FUNCTION_BLOCK IA_GBSD (* ISOBUS Adapter for Ground Based Speed and Distance (GBSD) *)
  (* Standard: ISO 11783-7; Classification: PGN 65097; Description: Copyright (c) 2024-2026 HR Agrartechnik GmbH This program and the accompanying materials are made available under the terms of the Eclipse Public License 2.0 which is available at https://www.eclipse.org/legal/epl-2.0/ SPDX-License-Identifier: EPL-2.0 *)
  (* Version 1.0, 2026-04-19, Franz Höpfinger, HR Agrartechnik GmbH, initial API and implementation (Adapter Wrapper for I_GBSD) *)
  PACKAGE isobus::tecu;
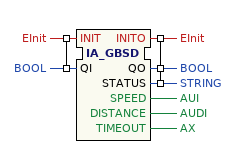
  EVENT_INPUT
    INIT : EInit WITH QI; (* Service Initialization *)
  END_EVENT
  EVENT_OUTPUT
    INITO : EInit WITH QO, STATUS; (* Initialization Confirm *)
  END_EVENT
  VAR_INPUT
    QI : BOOL; (* Event Input Qualifier *)
  END_VAR
  VAR_OUTPUT
    QO : BOOL; (* Event Output Qualifier *)
    STATUS : STRING;
  END_VAR
  PLUGS
    SPEED : adapter::types::unidirectional::AUI; (* Ground-based machine speed *)
    DISTANCE : adapter::types::unidirectional::AUDI; (* Ground-based machine distance *)
    TIMEOUT : adapter::types::unidirectional::AX; (* Timeout Status *)
  END_PLUGS
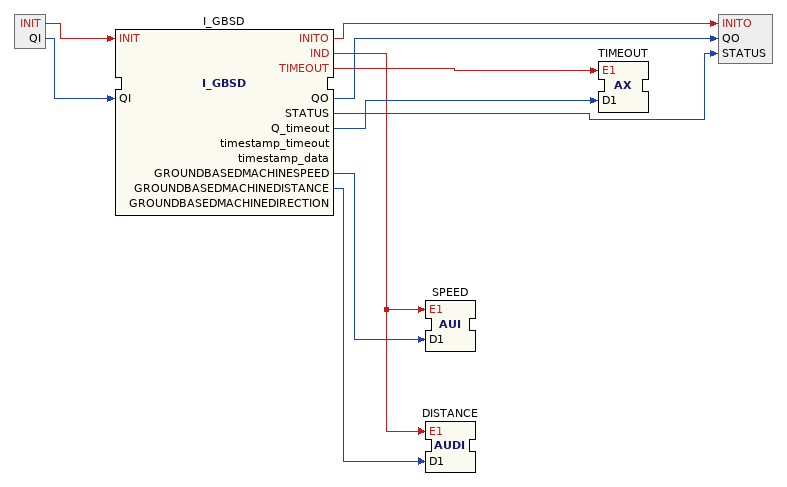
  FBS
    I_GBSD : isobus::tecu::I_GBSD;
  END_FBS
  EVENT_CONNECTIONS
    INIT TO I_GBSD.INIT;
    I_GBSD.INITO TO INITO;
    I_GBSD.IND TO DISTANCE.E1;
    I_GBSD.IND TO SPEED.E1;
    I_GBSD.TIMEOUT TO TIMEOUT.E1;
  END_CONNECTIONS
  DATA_CONNECTIONS
    QI TO I_GBSD.QI;
    I_GBSD.QO TO QO;
    I_GBSD.STATUS TO STATUS;
    I_GBSD.Q_timeout TO TIMEOUT.D1;
    I_GBSD.GROUNDBASEDMACHINESPEED TO SPEED.D1;
    I_GBSD.GROUNDBASEDMACHINEDISTANCE TO DISTANCE.D1;
  END_CONNECTIONS
END_FUNCTION_BLOCK
